// TIA Portal V19 export
DATA_BLOCK "HOUR_DB_3"   // DB56
// stored: InstanceOfName HOUR, InstanceOfType FB
"HOUR"
   // VAR_INPUT
   //    "SET TIME" : Int := 2;
   //    RESET : Bool;
   //    INPUT : Bool;
   // END_VAR
   // VAR_OUTPUT
   //    "PRESENT VALUE OF TIME" : Int;
   //    DONE : Bool;
   // END_VAR
   // VAR
   //    "TIMER 1" { S7_SetPoint := 'True'} : IEC_TIMER;
   // END_VAR
   // VAR RETAIN
   //    "COUNTER1 2" { S7_SetPoint := 'True'} : IEC_COUNTER;
   //    "COUNTER1 1" { S7_SetPoint := 'True'} : IEC_COUNTER;
   // END_VAR
   // VAR
   //    BIT { ExternalAccessible := 'False'; ExternalVisible := 'False'; ExternalWritable := 'False'} : Bool;
   // END_VAR
BEGIN
END_DATA_BLOCK
